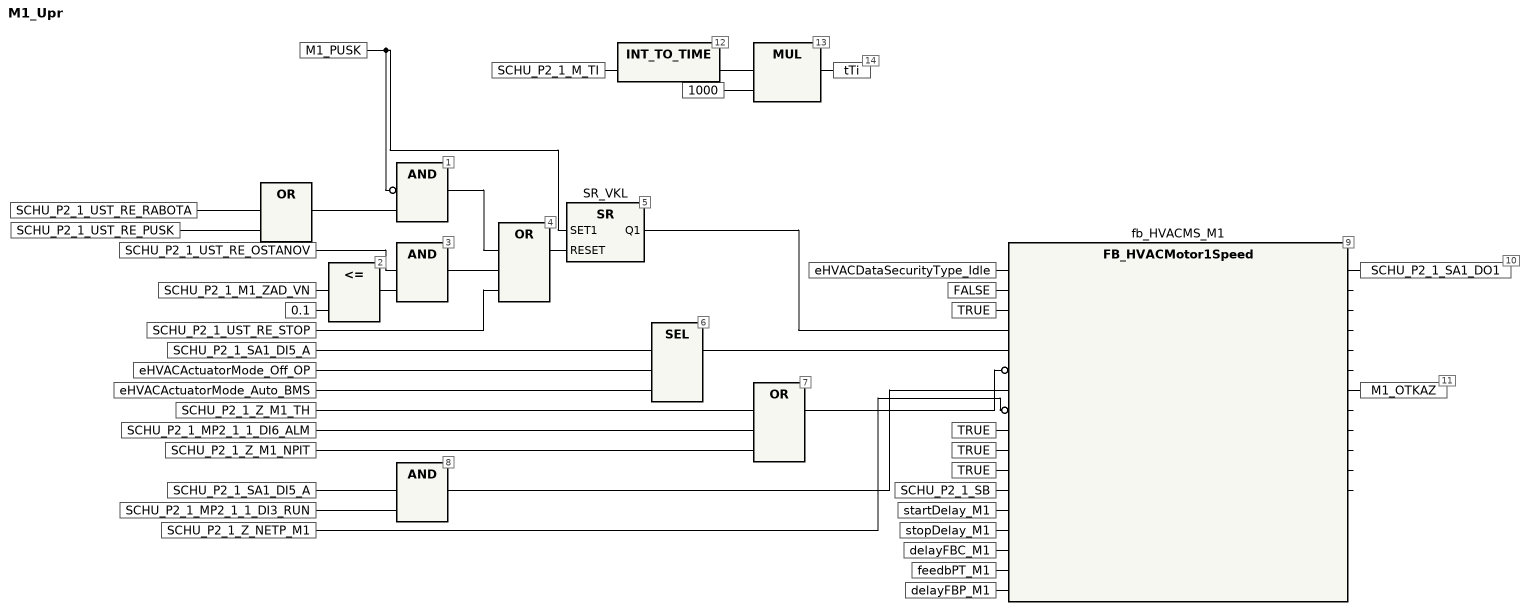
[picture p408: M1_Upr (CFC)]
_CFC_ (* Continuous Function Chart, elements in execution order *)
#0 OR(SCHU_P2_1_UST_RE_RABOTA, SCHU_P2_1_UST_RE_PUSK)
#1 AND(NOT M1_PUSK, #0)
#2 <=(SCHU_P2_1_M1_ZAD_VN, 0.1)
#3 AND(SCHU_P2_1_UST_RE_OSTANOV, #2)
#4 OR(#1, #3, SCHU_P2_1_UST_RE_STOP)
#5 SR_VKL:SR(SET1: M1_PUSK, RESET: #4)
#6 SEL(SCHU_P2_1_SA1_DI5_A, eHVACActuatorMode_Off_OP, eHVACActuatorMode_Auto_BMS)
#7 OR(SCHU_P2_1_Z_M1_TH, SCHU_P2_1_MP2_1_1_DI6_ALM, SCHU_P2_1_Z_M1_NPIT)
#8 AND(SCHU_P2_1_SA1_DI5_A, SCHU_P2_1_MP2_1_1_DI3_RUN)
#9 fb_HVACMS_M1:FB_HVACMotor1Speed(eHVACDataSecurityType_Idle, FALSE, TRUE, #5.Q1, #6, NOT #7, #8, NOT SCHU_P2_1_Z_NETP_M1, TRUE, TRUE, TRUE, SCHU_P2_1_SB, startDelay_M1, stopDelay_M1, delayFBC_M1, feedbPT_M1, delayFBP_M1)
#10 SCHU_P2_1_SA1_DO1 <= #9.out 1
#11 M1_OTKAZ <= #9.out 7
#12 INT_TO_TIME(SCHU_P2_1_M_TI)
#13 MUL(#12, 1000)
#14 tTi <= #13
_END_CFC_
END_PROGRAM

(* POU IM/M2_Upr, CFC *)
PROGRAM M2_Upr
VAR
	RS_M2: RS;

	startDelay_M2: TIME := T#0s;
	stopDelay_M2: TIME := T#0s;
	delayFBC_M2: TIME := T#30s;
	feedbPT_M2: TIME := T#120s;
	delayFBP_M2: TIME := T#30s;

	fb_HVACMS_M2: FB_HVACMotor1Speed;
	fb_HVACPIDC_M2: FB_HVACPIDCtrl;

	deadRange: REAL := 0.1;
	rKp: REAL := 1;
	tTi: TIME;
	tTv: TIME := T#0s;
	tTd: TIME := T#0s;
	direction: BOOL;
	rYMin: REAL;
	Dint_Ti: DINT;

	set: BOOL;
	reset: BOOL;
	resetContr: BOOL;
	RR_M2: RAMP_REAL;
	SR_START_REG: SR;
	RT_KOMVKL: R_TRIG;

	speedMotor: REAL;
	SR_VKL: SR;
	SCHU_P2_1_SA2_DI3_A: BOOL;
END_VAR
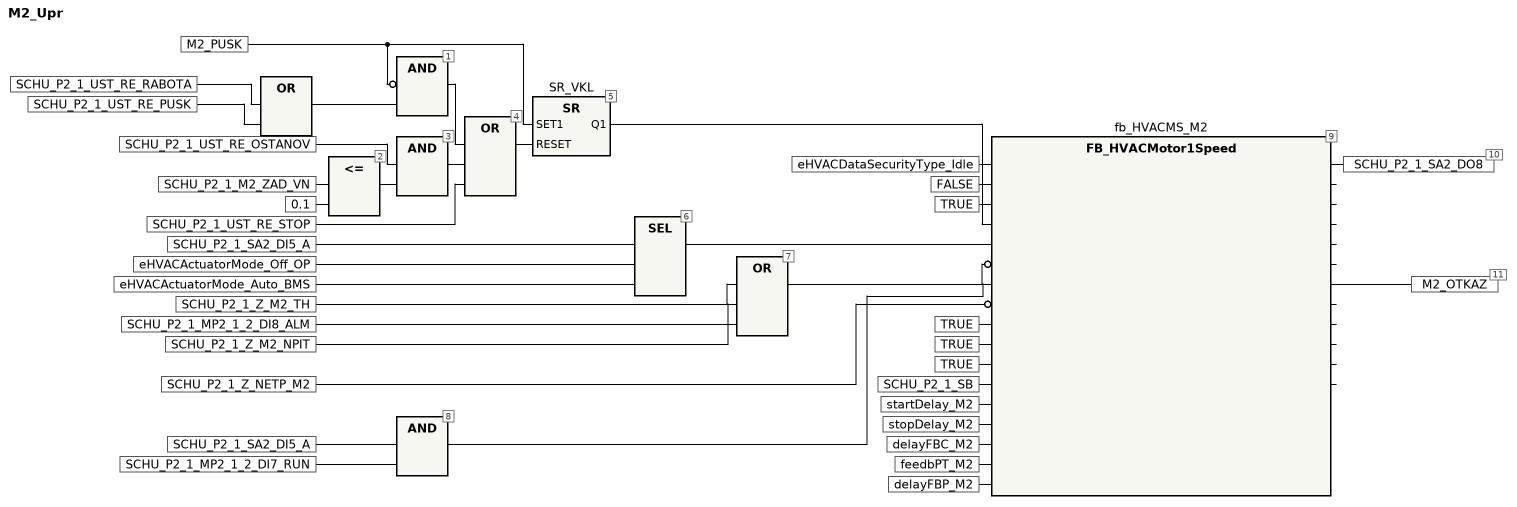
_CFC_ (* Continuous Function Chart, elements in execution order *)
#0 OR(SCHU_P2_1_UST_RE_RABOTA, SCHU_P2_1_UST_RE_PUSK)
#1 AND(NOT M2_PUSK, #0)
#2 <=(SCHU_P2_1_M2_ZAD_VN, 0.1)
#3 AND(SCHU_P2_1_UST_RE_OSTANOV, #2)
#4 OR(#1, #3, SCHU_P2_1_UST_RE_STOP)
#5 SR_VKL:SR(SET1: M2_PUSK, RESET: #4)
#6 SEL(SCHU_P2_1_SA2_DI5_A, eHVACActuatorMode_Off_OP, eHVACActuatorMode_Auto_BMS)
#7 OR(SCHU_P2_1_Z_M2_TH, SCHU_P2_1_MP2_1_2_DI8_ALM, SCHU_P2_1_Z_M2_NPIT)
#8 AND(SCHU_P2_1_SA2_DI5_A, SCHU_P2_1_MP2_1_2_DI7_RUN)
#9 fb_HVACMS_M2:FB_HVACMotor1Speed(eHVACDataSecurityType_Idle, FALSE, TRUE, #5.Q1, #6, NOT #7, #8, NOT SCHU_P2_1_Z_NETP_M2, TRUE, TRUE, TRUE, SCHU_P2_1_SB, startDelay_M2, stopDelay_M2, delayFBC_M2, feedbPT_M2, delayFBP_M2)
#10 SCHU_P2_1_SA2_DO8 <= #9.out 1
#11 M2_OTKAZ <= #9.out 7
_END_CFC_
END_PROGRAM

(* POU IM/PE_Upr, CFC *)
PROGRAM PE_Upr
VAR
	PE_PID: FB_HVACPIDCtrl;

	deadRange: REAL := 0.1;
	direction: BOOL;
	tTi: TIME;
	tTv: TIME;
	tTd: TIME;
	PE_PID_VKL: TON;
END_VAR
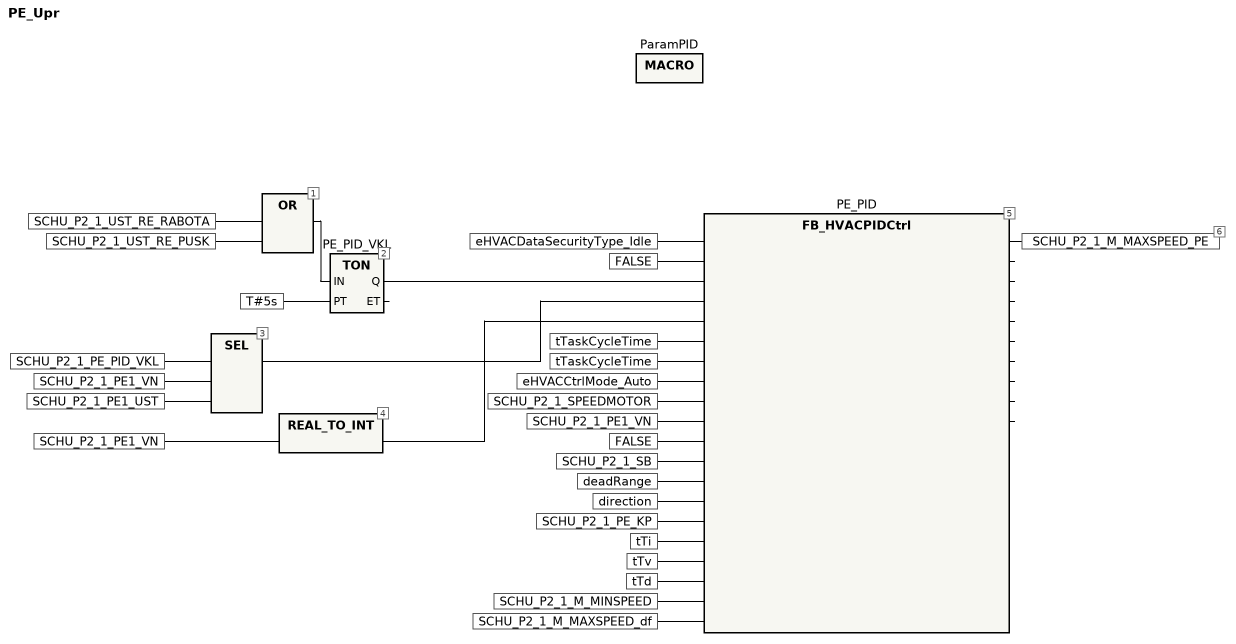
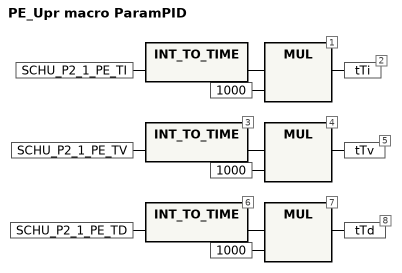
_CFC_ (* Continuous Function Chart, elements in execution order *)
#0 MACRO ParamPID()
	#1 INT_TO_TIME(SCHU_P2_1_PE_TI)
	#2 MUL(#1, 1000)
	#3 tTi <= #2
	#4 INT_TO_TIME(SCHU_P2_1_PE_TV)
	#5 MUL(#4, 1000)
	#6 tTv <= #5
	#7 INT_TO_TIME(SCHU_P2_1_PE_TD)
	#8 MUL(#7, 1000)
	#9 tTd <= #8
END_MACRO
#10 OR(SCHU_P2_1_UST_RE_RABOTA, SCHU_P2_1_UST_RE_PUSK)
#11 PE_PID_VKL:TON(IN: #10, PT: T#5s)
#12 SEL(SCHU_P2_1_PE_PID_VKL, SCHU_P2_1_PE1_VN, SCHU_P2_1_PE1_UST)
#13 REAL_TO_INT(SCHU_P2_1_PE1_VN)
#14 PE_PID:FB_HVACPIDCtrl(eHVACDataSecurityType_Idle, FALSE, #11.Q, #12, #13, tTaskCycleTime, tTaskCycleTime, eHVACCtrlMode_Auto, SCHU_P2_1_SPEEDMOTOR, SCHU_P2_1_PE1_VN, FALSE, SCHU_P2_1_SB, deadRange, direction, SCHU_P2_1_PE_KP, tTi, tTv, tTd, SCHU_P2_1_M_MINSPEED, SCHU_P2_1_M_MAXSPEED_df)
#15 SCHU_P2_1_M_MAXSPEED_PE <= #14.out 1
_END_CFC_
END_PROGRAM

(* POU IM/CHASTOTA_M1_M2, CFC *)
PROGRAM CHASTOTA_M1_M2
VAR
	RR: RAMP_REAL;
	SR_START_STER_REG: SR;
	SR_START_POV_REG: RS;
	RT_KOMVKL: R_TRIG;
	RT_KOMVKL_2: R_TRIG;
	RT_KOMVKL_1: R_TRIG;
	Zad_PE: TON;
	RS_RUCH: RS;
	V_RUCH: BOOL;
	TON_RUCH: TON;
	SCHU_P2_1_M_MAXSPEED_CH_OLD: REAL;
	SCHU_P2_1_PE1_UST_OLD: REAL;
	TON_STER_1: TON;
	TON_STER_2: TON;
	RT_PDK: R_TRIG;
	FT_PDK: F_TRIG;
END_VAR
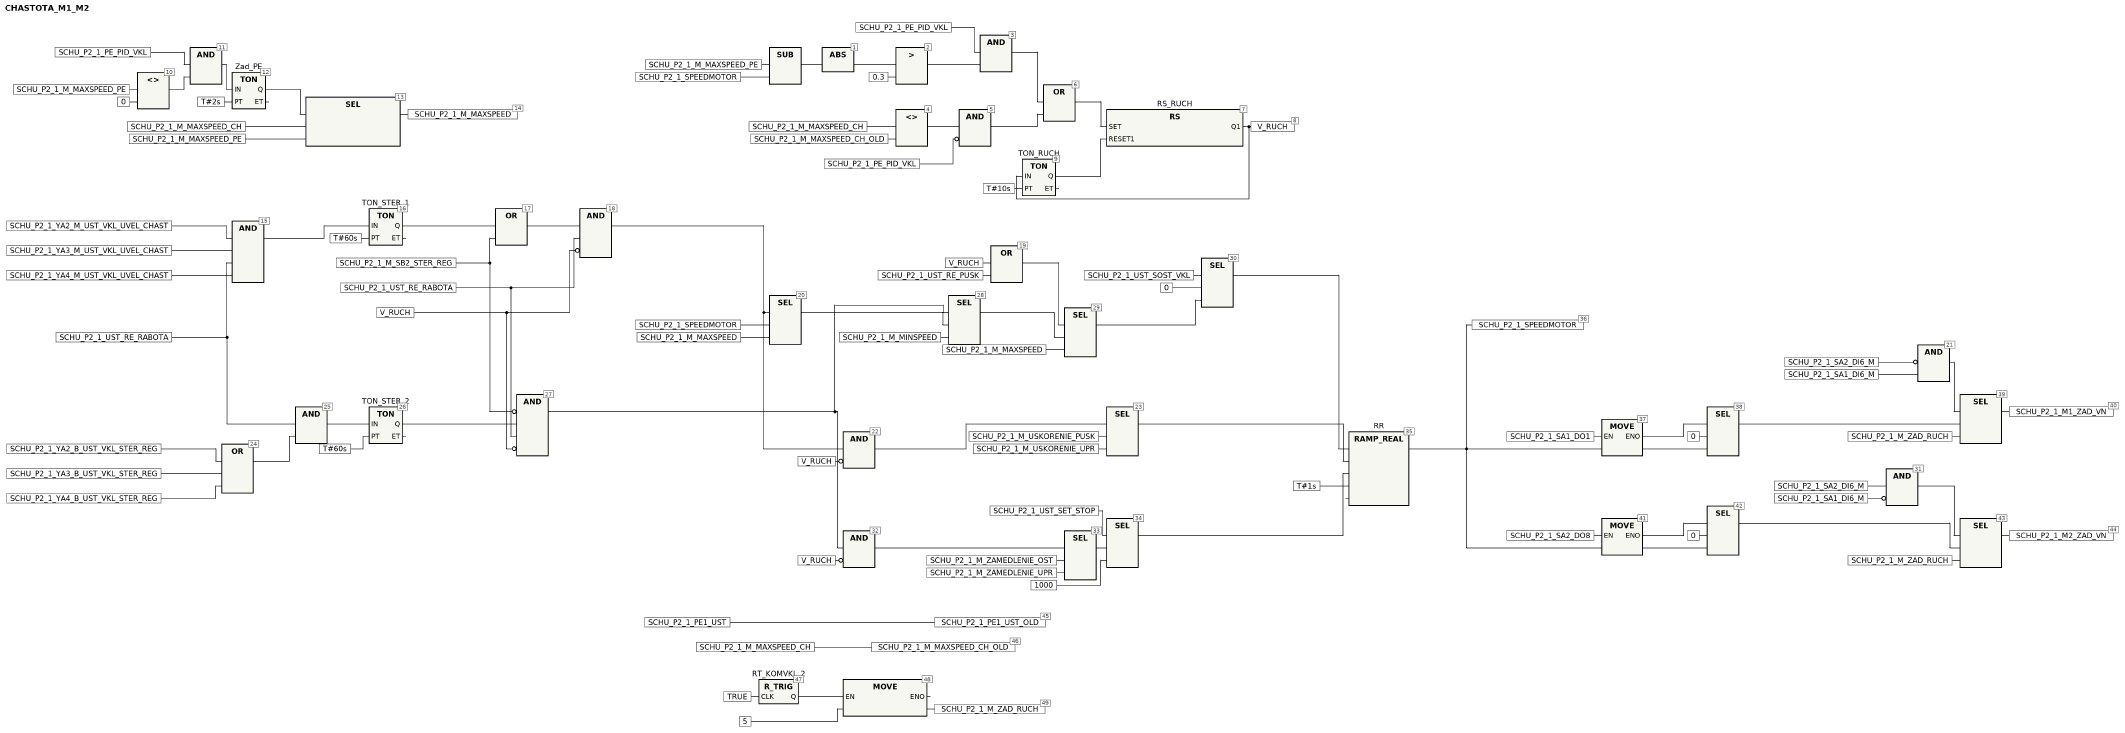
